(* PLC project Sin nombre, Desconocido Sin nombre 1 *)
(* stored: creationDateTime 2025-06-19T09:38:38, modificationDateTime 2025-06-19T10:10:40 *)

PROGRAM Main
  VAR
    iNivelTanque : INT;
    xBomba : BOOL;
    ArraySensores : ARRAY[0..3] OF INT;
    iSensor_1 : INT;
    iSensor_2 : INT;
    iSensor_3 : INT;
    iSensor_4 : INT;
    xAlarmaSobretemperatura : BOOL;
    i : INT;
    iTipoProducto : INT;
    rVelocidadCinta : REAL;
  END_VAR

            (*Sintaxis y Ejemplo - Sentencia IF*)
IF iNivelTanque < 30 THEN
    xBomba := TRUE;
  ELSE
    xBomba := FALSE;
END_IF;

(*Sintaxis y Ejemplo - Sentencia FOR*)
ArraySensores[0] := iSensor_1;
ArraySensores[1] := iSensor_2;
ArraySensores[2] := iSensor_3;
ArraySensores[3] := iSensor_4;

FOR i := 0 TO 3 BY 1 DO
  IF ArraySensores[i] > 80 THEN
    xAlarmaSobretemperatura := TRUE;
  END_IF;
END_FOR;

(*Sintaxis y Ejemplo - Sentencia CASE*)
CASE iTipoProducto OF
  1: rVelocidadCinta := 0.5; (*Producto liviano*)
  2: rVelocidadCinta := 1.0; (*Producto estándar*)
  3: rVelocidadCinta := 1.5; (*Producto pesado*)
  ELSE
    rVelocidadCinta := 0.0;
END_CASE;




          
END_PROGRAM

CONFIGURATION Config0
  RESOURCE Res0 ON PLC
    TASK task0(INTERVAL := T#20ms, PRIORITY := 0);
    PROGRAM instance0 WITH task0 : Main;
  END_RESOURCE
END_CONFIGURATION
